Staubli VAL3: checkCombo.pgx

program checkCombo(string& x_sResult)
  local num l_nCombo
begin

  for l_nCombo = 0 to size(lResult)-1

    if lResult[l_nCombo].sString == sCombo[0]+sCombo[1]

      x_sResult = lResult[l_nCombo].sString[1]
      return
    endIf

  endFor

  x_sResult = ""

end
